// SIMATIC S7-200 project (STEP 7-Micro/WIN), CPU 221 REL 01.10

ORGANIZATION_BLOCK 主程序:OB1
TITLE=程序注释
BEGIN
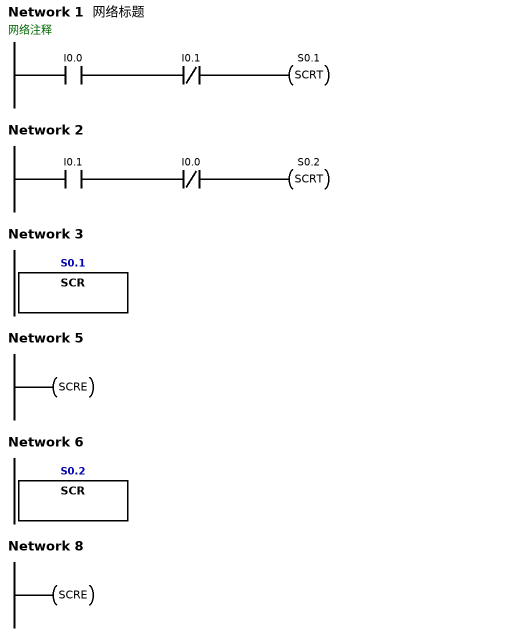
Network 1 // 网络标题
// 网络注释
// (network saved uncompiled; LAD cells follow)
// row 0: c0 -| |- I0.0  c1 -|/|- I0.1  c2 -(SCRT) S0.1
Network 2
// (network saved uncompiled; LAD cells follow)
// row 0: c0 -| |- I0.1  c1 -|/|- I0.0  c2 -(SCRT) S0.2
Network 3
// (network saved uncompiled; LAD cells follow)
// row 0: c0 [SCR S0.1 ]
Network 5
// (network saved uncompiled; LAD cells follow)
// row 0: c0 -(SCRE)
Network 6
// (network saved uncompiled; LAD cells follow)
// row 0: c0 [SCR S0.2 ]
Network 8
// (network saved uncompiled; LAD cells follow)
// row 0: c0 -(SCRE)
END_ORGANIZATION_BLOCK
